FUNCTION_BLOCK FB_DecodeCanRxMessage
VAR_INPUT
	RxMessage: CANQUEUE;
END_VAR
VAR_OUTPUT
	CobId: UINT;
	BytesReceived: UINT;
	arrDataReceived: CANMESSAGE;
END_VAR

BytesReceived := SHR((SHL(RxMessage.CobId,12)),12);
Cobid := SHR(rxMessage.CobId,5);
arrDataReceived := RxMessage.data;

END_FUNCTION_BLOCK

(* stored: Version 1.1.0.1, ProductVersion 3.1.0.23
   POU FB_DecodeCanRxMessage: Id {04e48716-0c9d-4f13-885d-bf169472b28d} *)
